Universal Robots PolyScope program: L02_pose.urp

Program L02_pose (installation=default directory=/programs createdIn=5.9.1.1031110 lastSavedIn=5.9.1.1031110 robotSerialNumber=20195501059)
Calibrated DH parameters: a=[0.000146, -0.418764, -0.053981, 0.000058, -0.000023, 0]; d=[0.162545, 37.319448, -206.067439, 168.881546, 0.09955, 0.099464]; alpha=[1.57004, -0.001979, 0.002304, 1.570607, -1.57066, 0]; deltaTheta=[0, -0.174616, -1.258233, 1.432844, -0.000001, 0]
Robot Program (runOnlyOnce=true)
  p01_p := get_actual_tcp_pose()
  MoveL speed 250 mm/s, acceleration 1200 mm/s^2 (useActiveTCP=true) feature=Base
    Waypoint Waypoint (Variable): variable=p01_p
    MoveDirectionNode (selectedDirection=XPlus)
      Until DISTANCE (allowActions=true deceleration=3 distanceNodeType=STOP) Distance=0.1; motionParameters(blendRadius=0)
        p02_p := get_actual_tcp_pose()
    Waypoint Waypoint (Variable): variable=p01_p
    MoveDirectionNode (selectedDirection=YPlus)
      Until DISTANCE (allowActions=true deceleration=3 distanceNodeType=STOP) Distance=0.1; motionParameters(blendRadius=0)
        p03_p := get_actual_tcp_pose()
    Waypoint Waypoint (Variable): variable=p01_p
    MoveDirectionNode (selectedDirection=ZPlus)
      Until DISTANCE (allowActions=true deceleration=3 distanceNodeType=STOP) Distance=0.1; motionParameters(blendRadius=0)
        p04_p := get_actual_tcp_pose()
    Waypoint Waypoint (Variable): variable=p01_p
